{attribute 'qualified_only'}
{attribute 'to_string'}
TYPE E_ConveyorMode :
(
	Auto := 0,
	Manual
) UINT;
END_TYPE

(* stored: Version 1.1.0.1, ProductVersion 3.1.4026.17
   DUT E_ConveyorMode: Id {772fa306-58c0-4b4d-a2a5-1fd856cb2e54} *)
